FUNCTION F_Time2lrMinute : lreal
VAR_INPUT
	t : TIME;
END_VAR
VAR
END_VAR

F_Time2lrMinute := time_to_lreal(t)*0.001*0.01666666667; // *0.001*0.01666666667 = /1000/60

END_FUNCTION

(* stored: Version 1.1.0.1, ProductVersion 3.1.4024.12
   POU F_Time2lrMinute: Id {043a305d-24f1-489d-aae5-21da2ce7d15b}, SpecialFunc None *)
